// Entry point for the Sift Client. This function block must be initialized successfully
// first before using any of the other services. The function block begins initialization
// on the rising edge of bExecute and completes initialization when bBusy goes low.
FUNCTION_BLOCK FB_SiftClient
VAR_INPUT
	sSiftProxyHost : T_IPv4Addr := GVL_SIFT.SIFT_PROXY_DEFAULT_HOST;
	nSiftProxyPort : UINT       := GVL_SIFT.SIFT_PROXY_DEFAULT_LISTEN_PORT;
	sLogDir : STRING(255);
	
	sGrpcUri : STRING(255);
	sApiKey : STRING(255);
	
	pJsonBuffer : POINTER TO BYTE;
	pJbLength : UDINT;
	
	bExecute : BOOL;
	bStop : BOOL;
END_VAR

VAR_OUTPUT
	hSiftClient : T_SiftClient;
	bBusy : BOOL;
	bError : BOOL;
	nErrId : UDINT;
	nErrMsg : STRING(255);
END_VAR

VAR
    fbAuth : FB_AuthenticateService;	
	fbStartSiftProxy : NT_StartProcess;
	fbGetLocalAmsNetID : FB_GetLocalAmsNetId;
	fbFormat : FB_FormatString;
	nAttempts : UINT;
	startDelay : TON;
	
	eState : (
		IDLE, 
		CLOSE_ALL, 
		CLOSE_ALL_WAIT, 
		CONNECT, 
		CONNECT_WAIT, 
		GET_LOCAL_AMD_NET_ID,
		GET_LOCAL_AMD_NET_ID_WAIT,
		START_SIFT_PROXY, 
		START_SIFT_PROXY_DELAY,
		START_SIFT_PROXY_WAIT,
		AUTHENTICATE,
		AUTHENTICATE_WAIT,
		SUCCESS, 
		FAILURE,
		STOP,
		STOP_WAIT,
	) := IDLE;
END_VAR

CASE eState OF
	IDLE:
	    bBusy := FALSE;
		IF bExecute THEN
			eState := CLOSE_ALL;
		ELSIF bStop THEN
			eState := STOP;
		END_IF

	CLOSE_ALL:
		bBusy := TRUE;
		bError := FALSE;
		hSiftClient.fbCloseAll(bExecute := TRUE);
		nAttempts := 0;
		eState := CLOSE_ALL_WAIT;
		
	CLOSE_ALL_WAIT:
		bBusy := TRUE;
		bError := FALSE;
		hSiftClient.fbCloseAll(bExecute := FALSE);
		
		IF hSiftClient.fbCloseAll.bBusy THEN
			RETURN;
		ELSIF hSiftClient.fbCloseAll.bError THEN
			nErrId := hSiftClient.fbCloseAll.nErrId;
			eState := FAILURE;
			nErrMsg := 'Failed to call FB_CloseAll';
			RETURN;
		END_IF
		eState := CONNECT;

	CONNECT:
		bBusy := TRUE;
		bError := FALSE;
		hSiftClient.sHost := sSiftProxyHost;
		hSiftClient.nPort := nSiftProxyPort;
		hSiftClient.sApiKey := sApiKey;
		hSiftClient.sGrpcUri := sGrpcUri;
		
		IF pJsonBuffer = 0 THEN
			nErrId := GVL_SIFT.NULL_JSON_POINTER;
			eState := FAILURE;
			RETURN;
		END_IF
		hSiftClient.pJsonBuffer := pJsonBuffer;
		hSiftClient.pJbLength := pJbLength;
		
		hSiftClient.fbConnect(sRemoteHost := sSiftProxyHost, 
						      nRemotePort := nSiftProxyPort, 
							  bExecute := TRUE,
							  tTimeout := T#1S);
		
		nAttempts := nAttempts + 1;
		IF nAttempts >= 3 THEN
			nErrId := GVL_SIFT.SIFT_PROXY_FAILED_TO_START;
			nErrMsg := 'Failed to connect to sift-proxy';
			eState := FAILURE;
			RETURN;
		END_IF
		
		eState := CONNECT_WAIT;
		
	CONNECT_WAIT:
		bBusy := TRUE;
		bError := FALSE;
		hSiftClient.fbConnect(bExecute := FALSE);
		
		IF hSiftClient.fbConnect.bBusy THEN
			RETURN;
		ELSIF hSiftClient.fbConnect.bError THEN
			nErrId := hSiftClient.fbConnect.nErrId;
			eState := GET_LOCAL_AMD_NET_ID;
			RETURN;
		END_IF
		eState := AUTHENTICATE;
		
	GET_LOCAL_AMD_NET_ID:
		bBusy := TRUE;
		bError := FALSE;
		fbGetLocalAmsNetID(bExecute := TRUE);
		eState := GET_LOCAL_AMD_NET_ID_WAIT;
		
	GET_LOCAL_AMD_NET_ID_WAIT:
		bBusy := TRUE;
		bError := FALSE;
		fbGetLocalAmsNetID(bExecute := FALSE);
		
		IF fbGetLocalAmsNetID.bBusy THEN
			RETURN;
		ELSIF fbGetLocalAmsNetID.bError THEN
			nErrId := fbGetLocalAmsNetID.nErrId;
			nErrMsg := 'Failed to get local AmsNetId';
			eState := FAILURE;
			RETURN;
		END_IF
		eState := START_SIFT_PROXY;

	START_SIFT_PROXY:
		bBusy := TRUE;
		bError := FALSE;
		IF sGrpcUri = '' THEN
			nErrId := GVL_SIFT.INVALID_GRPC_URI;
			nErrMsg := 'GRPC URI not set';
			eState := FAILURE;
			RETURN;
		END_IF
		IF sApiKey = '' THEN
			nErrId := GVL_SIFT.INVALID_API_KEY;
			nErrMsg := 'API Key not set';
			eState := FAILURE;
			RETURN;
		END_IF
		IF sLogDir = '' THEN
			nErrId := GVL_SIFT.INVALID_LOG_DIR;
			nErrMsg := 'Log directory not set';
			eState := FAILURE;
			RETURN;
		END_IF
				
		fbFormat(
			sFormat := GVL_SIFT.SIFT_PROXY_CMD_ARGS, 
			arg1 := F_STRING(sLogDir),
			arg2 := F_UINT(nSiftProxyPort), 
			arg3 := F_STRING(sGrpcUri), 
			arg4 := F_STRING(sApiKey),
		);
		IF fbFormat.bError THEN
			nErrId := fbFormat.nErrId;
			nErrMsg := 'Failed to create sift-proxy command';
			eState := FAILURE;
		END_IF
		
		fbStartSiftProxy(
			NetId:=fbGetLocalAmsNetID.AddrString,
			PATHSTR:=SiftClientParameters.START_SIFT_PROXY_PATH, 
			COMNDLINE:=fbFormat.sOut,
			START := TRUE,
		);

		eState := START_SIFT_PROXY_WAIT;
				
	START_SIFT_PROXY_WAIT:
		bBusy := TRUE;
		bError := FALSE;
		fbStartSiftProxy(START := FALSE);
		
		IF fbStartSiftProxy.BUSY THEN
			RETURN;
		ELSIF fbStartSiftProxy.ERR THEN
			nErrId := fbStartSiftProxy.ERRID;
			nErrMsg := 'Failed to start sift-proxy';
			eState := FAILURE;
			RETURN;
		END_IF

		startDelay(IN:=FALSE);
		startDelay(IN:=TRUE, PT:=GVL_SIFT.SIFT_PROXY_START_DELAY);
		
		eState := START_SIFT_PROXY_DELAY;

	START_SIFT_PROXY_DELAY:
		bBusy := TRUE;
		bError := FALSE;
		
		startDelay();
		IF NOT startDelay.Q THEN
			RETURN;
		END_IF
		
		eState := CONNECT;
		
	AUTHENTICATE:
		bBusy := TRUE;
		bError := FALSE;
		fbAuth(hSiftClient:=hSiftClient, bExecute:=TRUE);
		eState := AUTHENTICATE_WAIT;
		
	AUTHENTICATE_WAIT:
		bBusy := TRUE;
		bError := FALSE;
		fbAuth(bExecute:=FALSE);
		
		IF fbAuth.bBusy THEN
			RETURN;
		ELSIF fbAuth.bError THEN
			nErrId := fbAuth.nErrId;
			nErrMsg := 'Failed to authenticate';
			eState := FAILURE;
			RETURN;
		END_IF
		eState := SUCCESS;
		
	SUCCESS:
		bBusy := FALSE;
		bError := FALSE;
		eState := IDLE;
		
	FAILURE:
		bBusy := FALSE;
		bError := TRUE;
		eState := IDLE;
		
	STOP:
		bBusy := TRUE;
		bError := FALSE;
		hSiftClient.fbCloseAll(bExecute := TRUE);
		eState := STOP_WAIT;
		
	STOP_WAIT:
		bBusy := TRUE;
		bError := FALSE;
		hSiftClient.fbCloseAll(bExecute := FALSE);
		
		IF hSiftClient.fbCloseAll.bBusy THEN
			RETURN;
		ELSIF hSiftClient.fbCloseAll.bError THEN
			nErrId := hSiftClient.fbCloseAll.nErrId;
			nErrMsg := 'Failed to call FB_CloseAll';
			eState := FAILURE;
			RETURN;
		END_IF
		eState := IDLE;
END_CASE

END_FUNCTION_BLOCK

(* stored: Version 1.1.0.1
   POU FB_SiftClient: Id {4caab956-b0cf-47ee-89e4-4108cb730320}, SpecialFunc None *)
